// TIA Portal V19 export
TYPE "LEXCHANGETRAY_typePlasticWorkStationIoSignalControlNode"
// reset: Bool
// monitoring: LEXCHANGETRAY_typePlasticWorkStationIoSignalContronNodeMonitoring
// stored: Access Published
   STRUCT
      reset : Bool;
      monitoring { S7_SetPoint := 'True'} : "LEXCHANGETRAY_typePlasticWorkStationIoSignalContronNodeMonitoring";
   END_STRUCT;
END_TYPE
